INTERFACE IStirControl

PROPERTY pSetpoint : LREAL
GET
END_GET
END_PROPERTY

METHOD StirControl : LREAL
VAR_INPUT
	i : INT;
END_VAR
END_METHOD

END_INTERFACE

(* stored: Version 1.1.0.1, ProductVersion 3.1.4024.9
   Itf IStirControl: Id {1e704fb4-6e47-4c22-9b93-334a91c88fa2}
   Property pSetpoint: Id {12ecc515-0b9d-48e5-b673-fddecff709c8}
   Get Get: Id {b6554fe7-be67-4ec9-9e0d-011930fc55ee}
   Method StirControl: Id {645c9bcd-be6f-404b-b326-840963d81083} *)
